FUNCTION_BLOCK Section5Ctrl (* Basic Function Block Type *)
  (* Standard: 61499-2 *)
  (* Version 0.0, 5/27/2018, MIA, nxtControl GmbH, Template *)
  PACKAGE Main;
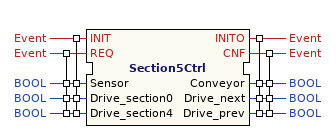
  EVENT_INPUT
    INIT WITH Sensor, Drive_section0, Drive_section4; (* Initialization Request *)
    REQ WITH Sensor, Drive_section0, Drive_section4; (* Normal Execution Request *)
  END_EVENT
  EVENT_OUTPUT
    INITO WITH Conveyor, Drive_next, Drive_prev; (* Initialization Confirm *)
    CNF WITH Conveyor, Drive_next, Drive_prev; (* Execution Confirmation *)
  END_EVENT
  VAR_INPUT
    Sensor : BOOL; (* Input event qualifier *)
    Drive_section0 : BOOL;
    Drive_section4 : BOOL;
  END_VAR
  VAR_OUTPUT
    Conveyor : BOOL; (* Output event qualifier *)
    Drive_next : BOOL;
    Drive_prev : BOOL;
  END_VAR
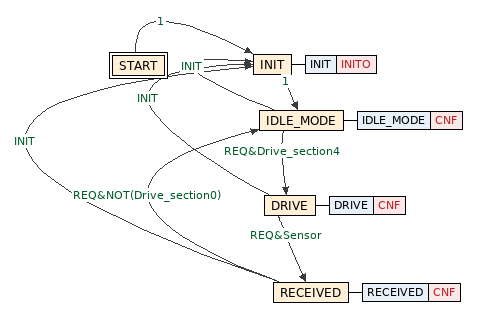
  EC_STATES
    START; (* Initial State *)
    INIT : INIT -> INITO; (* Initialization *)
    IDLE_MODE : IDLE_MODE -> CNF;
    DRIVE : DRIVE -> CNF;
    RECEIVED : RECEIVED -> CNF;
  END_STATES
  EC_TRANSITIONS
    START TO INIT := 1;
    INIT TO IDLE_MODE := 1;
    IDLE_MODE TO DRIVE := REQ&Drive_section4;
    DRIVE TO RECEIVED := REQ&Sensor;
    RECEIVED TO IDLE_MODE := REQ&NOT(Drive_section0);
    IDLE_MODE TO INIT := INIT;
    DRIVE TO INIT := INIT;
    RECEIVED TO INIT := INIT;
  END_TRANSITIONS
  ALGORITHM INIT IN ST: (* Initialization algorithm *)
;
Conveyor := FALSE;
Drive_prev := FALSE;
Drive_next := FALSE;
  END_ALGORITHM
  ALGORITHM IDLE_MODE IN ST:
;
Conveyor := FALSE;
Drive_prev := TRUE;
Drive_next := FALSE;
  END_ALGORITHM
  ALGORITHM DRIVE IN ST:
;
Conveyor := TRUE;
Drive_prev := TRUE;
Drive_next := FALSE;
  END_ALGORITHM
  ALGORITHM RECEIVED IN ST:
;
Conveyor := TRUE;
Drive_prev := FALSE;
Drive_next := TRUE;
  END_ALGORITHM
END_FUNCTION_BLOCK
